FUNCTION_BLOCK FB_Deadband_Auto
VAR_INPUT
	fClosedloopSignal	: LREAL;
	fVelref				: LREAL;
	fNeutral			: LREAL;
	fupperdeadband		: LREAL;
	flowerdeadband		: LREAL;
	
END_VAR
VAR_OUTPUT
	fDeadbandComp		: LREAL;
END_VAR
VAR
END_VAR

IF fVelref > 0.01 THEN
	fDeadbandComp := LIMIT(fNeutral,fupperdeadband + fClosedloopSignal,1.0);
ELSIF fVelref < -0.01 THEN
	fDeadbandComp := LIMIT(0.1,flowerdeadband + fClosedloopSignal,fNeutral); //Kanskje minus her men tror input blir - så da blir det fikset
ELSE
	fDeadbandComp := LIMIT(-1.0,fNeutral,1.0);
END_IF

END_FUNCTION_BLOCK

(* stored: Version 1.1.0.1
   POU FB_Deadband_Auto: Id {6ce62f62-654a-48a7-991c-330136cf95a0}, SpecialFunc None *)
